TYPE T_JANSSEN_CTRL EXTENDS T_RS_BASE_CTRL :
STRUCT
	// Arrays of structures for Configuration and Control commands.
	// Note that only one positioner is handled in each monitoring cycle.
	{attribute 'OPC.UA.DA' := '0'}
	cmdList:			ARRAY [0..15]	OF T_JANSSEN_COMMAND;	// List of up to 16 Commands per channel
	
END_STRUCT
END_TYPE

(* stored: Version 1.1.0.1, ProductVersion 3.1.4024.12
   DUT T_JANSSEN_CTRL: Id {1e560b52-4c68-45d1-adae-5872a1d74c82} *)
